PROGRAM DemandedSpeedCalculator
VAR
END_VAR

END_PROGRAM

(* stored: Version 1.1.0.1, ProductVersion 3.1.4022.16
   POU DemandedSpeedCalculator: Id {38457ad0-6fb8-4aa3-a566-b0aa09b9588e}, SpecialFunc None *)
